PROGRAM prgSafetyMain
VAR
END_VAR

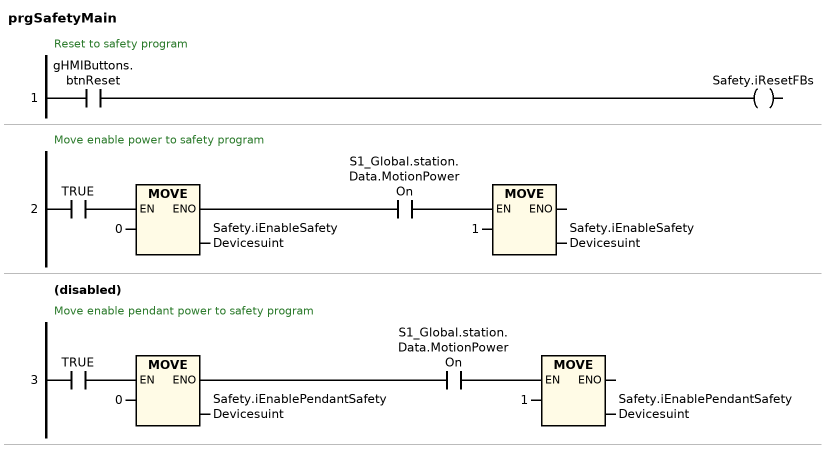
// NETWORK 1
// Reset to safety program
Safety.iResetFBs := gHMIButtons.btnReset;

// NETWORK 2
// Move enable power to safety program
Safety.iEnableSafetyDevicesuint := 0;
IF TRUE AND S1_Global.station.Data.MotionPowerOn THEN Safety.iEnableSafetyDevicesuint := 1; END_IF

// NETWORK 3 (disabled)
// Move enable pendant power to safety program
// Safety.iEnablePendantSafetyDevicesuint := 0;
// IF TRUE AND S1_Global.station.Data.MotionPowerOn THEN Safety.iEnablePendantSafetyDevicesuint := 1; END_IF

END_PROGRAM

(* stored: Version 1.1.0.1, ProductVersion 3.1.4024.12
   POU prgSafetyMain: Id {131003ea-c5f7-4052-9a6a-c5b277ac1841}, SpecialFunc None *)
